// TIA Portal project "Custom_end_assignment" (V17)

(* hardware
DEVICE "S7-1200 station_1"  S7-1200 Station
   slot 0: "Rack_0"  S7-1200 Rack  Rack  V1.0
   slot 1: "PLC_1"  CPU 1215C AC/DC/Rly  6ES7 215-1BG40-0XB0  V4.5
DEVICE "HMI_1"  KTP700 Basic PN
   slot 0: "HMI_1"  KTP700 Basic PN  6AV2 123-2GB03-0AX0  17.0.0.0
   slot 1: "HMI_RT_1"  KTP700 Basic PN  6AV2 123-2GB03-0AX0  17.0.0.0
   slot 5: "HMI_1.IE_CP_1"  PROFINET Interface  17.0.0.0
      slot 1: "PROFINET Interface_1"  PROFINET Interface
         slot 1: "Port_1"  Port
*)

// ===== PLC "PLC_1"  CPU 1215C AC/DC/Rly =====

VAR_GLOBAL   // PLC tag table "Default tag table"
   "System_Byte" AT %MB1 : Byte;
   "FirstScan" AT %M1.0 : Bool;
   "DiagStatusUpdate" AT %M1.1 : Bool;
   "AlwaysTRUE" AT %M1.2 : Bool;
   "AlwaysFALSE" AT %M1.3 : Bool;
   "Clock_Byte" AT %MB0 : Byte;
   "Clock_10Hz" AT %M0.0 : Bool;
   "Clock_5Hz" AT %M0.1 : Bool;
   "Clock_2.5Hz" AT %M0.2 : Bool;
   "Clock_2Hz" AT %M0.3 : Bool;
   "Clock_1.25Hz" AT %M0.4 : Bool;
   "Clock_1Hz" AT %M0.5 : Bool;
   "Clock_0.625Hz" AT %M0.6 : Bool;
   "Clock_0.5Hz" AT %M0.7 : Bool;
END_VAR

VAR_GLOBAL   // PLC tag table "Hardware_I_O_Tags"
   "i_DR1_FlowSensorWaste" AT %I0.0 : Bool;
   "i_DR2_FlowSensorProduct" AT %I0.1 : Bool;
   "i_DR3_FlowSensorCocoa" AT %I0.2 : Bool;
   "i_DR4_FlowSensorSugar" AT %I0.3 : Bool;
   "i_RP_Start" AT %I0.4 : Bool;
   "i_RP_CocoaMinus" AT %I0.5 : Bool;
   "i_RP_CocoaPlus" AT %I0.6 : Bool;
   "i_RP_SugarMinus" AT %I0.7 : Bool;
   "i_RP_SugarPlus" AT %I1.0 : Bool;
   "i_RP_AllMilk" AT %I1.1 : Bool;
   "i_CP_CleanMinus" AT %I1.2 : Bool;
   "i_CP_BatchesMinus" AT %I1.3 : Bool;
   "i_CP_BatchesPlus" AT %I1.4 : Bool;
   "i_CP_1Batch" AT %I1.5 : Bool;
   "i_Tank_HeaterFeedback" AT %I8.0 : Bool;
   "i_Tank_LevelLow" AT %I8.1 : Bool;
   "i_Tank_LevelMiddle" AT %I8.2 : Bool;
   "i_Tank_LevelHigh" AT %I8.3 : Bool;
   "i_CP_Start" AT %I8.4 : Bool;
   "o_Tank_ValveWaste" AT %Q0.0 : Bool;
   "o_Tank_ValveProduct" AT %Q0.1 : Bool;
   "o_Tank_ValveCocoa" AT %Q0.2 : Bool;
   "o_Tank_ValveSugar" AT %Q0.3 : Bool;
   "o_Tank_ValveMilk" AT %Q0.4 : Bool;
   "o_Tank_ValveWater" AT %Q0.5 : Bool;
   "o_RP_Started_LED" AT %Q0.6 : Bool;
   "o_RP_Cocoa_LED" AT %Q0.7 : Bool;
   "o_RP_Sugar_LED" AT %Q1.0 : Bool;
   "o_RP_AllMilk_LED" AT %Q1.1 : Bool;
   "o_Tank_LevelEmpty_LED" AT %Q12.0 : Bool;
   "o_Tank_LevelLow_LED" AT %Q12.1 : Bool;
   "o_Tank_LevelMiddle_LED" AT %Q12.2 : Bool;
   "o_Tank_LevelHigh_LED" AT %Q12.3 : Bool;
   "o_Tank_Heater" AT %Q12.4 : Bool;
   "o_Tank_Mixer" AT %Q12.5 : Bool;
   "ai_Tank_Level" AT %IW64 : Int;
   "TankLevelScaledValue" AT %MD0 : Real;
   "ai_Tank_Temperature" AT %IW66 : Int;
   "TankTemperatureScaledValue" AT %MD4 : Real;
END_VAR

DATA_BLOCK "DB_MixerTank"   // DB2
{ S7_Optimized_Access := 'TRUE' }
VERSION : 0.1
   VAR
      i_FlowRate : Real := 1.0;
      ai_TankVolume : Real;
      ScaledTankVolume : Real;
      i_StartProcess : Bool;
      i_EmergencyStopOK : Bool;
      BoosterPumpMultiplier : Real := 5.0;
      MixerTankCapacity : Real := 500.0;
   END_VAR
BEGIN
END_DATA_BLOCK

// folder: 01_Communication/HumanMachineInterface

DATA_BLOCK "DB_MixerTankSystem"   // DB15
{ S7_Optimized_Access := 'TRUE' }
VERSION : 0.1
   VAR
      Valve1 : Bool;   // 0= closed, 1 = open
      Valve2 : Bool;   // 0= closed, 1 = open
      Valve3 : Bool;   // 0= closed, 1 = open
      FlowValve1 : Real;   // The amount of flow through valve 1 (input), Max 10 in normal mode
      FlowValve2 : Real;   // The amount of flow through valve 2 (input) Max 10 in normal mode
      FlowValve3 : Real;   // The amount of flow through valve 3 (output) Max 10 in normal mode
      MotorFlowValve1 : Bool;   // 0 = off / 1 = on
      MotorFlowValve2 : Bool;   // 0 = off / 1 = on
      MotorFlowValve3 : Bool;   // 0 = off / 1 = on
      MotorMixer : Bool;   // 0 = off / 1 = on
      TimerMotorMixer : Time;   // Timer Motor mixer is on (s)
      SystemStatusTank : Int;   // user defined type
      SensorTankVolumeHigh : Bool;   // sensor tank volume high
      SensorTankVolumeMiddle : Bool;   // sensor tank volume middle
      SensorTankVolumeLow : Bool;   // sensor tank volume low
      SensorBottleClamped : Bool;   // bottle is clamped by cilinder (1 = clamped / 0 = not clamped)
      Temperature : Real;
      ModeTemperature : Bool;   // 0= Celcius / 1= Fahrenheit
      Heating : Bool;   // 0 = off / 1 = on
      VolumeTank : Real;   // Total volume in the tank (MAX500L)
      NumberOfBottles : Int;   // Number of Bottles that are filled (each bottle 250 mL)
      "Status System" : String;   // defines message as 'fill bottle', valve1 open, valve 2 open
      Startbutton : Bool;
      StopButton : Bool;
   END_VAR
BEGIN
END_DATA_BLOCK

DATA_BLOCK "DB_BottleConveyer"   // DB16
{ S7_Optimized_Access := 'TRUE' }
VERSION : 0.1
   VAR
      A1 : Bool;   // Main switch bottle conveyor
      A2 : Bool;   // Automatic start bottle conveyor
      M1 : Bool;   // On/Off bottle conveyor
      B1 : Bool;   // Sensor infeed bottle conveyor
      B2 : Bool;   // Sensor bottle present filling nozzle
      B3 : Bool;   // Sensor bottle present bottlecheck
      B4 : Bool;   // Sensor bottle filled bottlecheck
      B5 : Bool;   // Sensor outfeed bottle conveyor
      P1 : Bool;   // Status servo bottle clamping
      P2 : Bool;   // Status servo cap positioning
   END_VAR
BEGIN
END_DATA_BLOCK

// folder: 01_Communication/System1

DATA_BLOCK "PC_Communication_Tags_Sys1"   // DB100
{ S7_Optimized_Access := 'TRUE' }
VERSION : 0.1
   VAR
      ServoPower : Bool;   // On/Off: On the HMI there is a button what switches on and off the power of the connected Servo
      RunState : Bool;   // This tag is True when the state of the whole system is 'Run'
      StopState : Bool;   // This tag is True when the state of the whole system is 'Stop'
      EnableReceiveCommands : Bool;   // On/Off: On the HMI there is a button what switches on and off the communication service
      MotorActiveFwd : Bool;   // This tag is True when the connected Servo is moving forward
      MotorActiveRev : Bool;   // This tag is True when the connected Servo is moving reverse
      SystemReadyServoActions : Bool;   // Only when all conditions are met (like described in the assessment document) this tag is True
      StartServoActions : Bool;   // When this tag is True, the Servo sequence may start "at the other side"
      ServoActionsFinished : Bool;   // When the actions to be executed for the connected Servo are finished, this tag is True
      BottlePresentRobot : Bool;   // This tag is True when a bottle is present at the robot
      BottleFilled : Bool;   // This tag is True when a bottle is filled
      BottleNotFilled : Bool;   // This tag is True when a bittle is not filled
      HeartBeat : Bool;   // This is a "heart beat" signal what is toggeling state in 0.5Hz frequency
   END_VAR
BEGIN
END_DATA_BLOCK

// folder: 01_Communication/System2

DATA_BLOCK "PC_Communication_Tags_Sys2"   // DB101
{ S7_Optimized_Access := 'TRUE' }
VERSION : 0.1
   VAR
      ServoPower : Bool;   // On/Off: On the HMI there is a button what switches on and off the power of the connected Servo
      RunState : Bool;   // This tag is True when the state of the whole system is 'Run'
      StopState : Bool;   // This tag is True when the state of the whole system is 'Stop'
      EnableReceiveCommands : Bool;   // On/Off: On the HMI there is a button what switches on and off the communication service
      MotorActiveFwd : Bool;   // This tag is True when the connected Servo is moving forward
      MotorActiveRev : Bool;   // This tag is True when the connected Servo is moving reverse
      SystemReadyServoActions : Bool;   // Only when all conditions are met (like described in the assessment document) this tag is True
      StartServoActions : Bool;   // When this tag is True, the Servo sequence may start "at the other side"
      ServoActionsFinished : Bool;   // When the actions to be executed for the connected Servo are finished, this tag is True
      BottlePresentRobot : Bool;   // This tag is True when a bottle is present at the robot
      BottleFilled : Bool;   // This tag is True when a bottle is filled
      BottleNotFilled : Bool;   // This tag is True when a bittle is not filled
      HeartBeat : Bool;   // This is a "heart beat" signal what is toggeling state in 0.5Hz frequency
   END_VAR
BEGIN
END_DATA_BLOCK

// folder: 02_Unit_MixerTank

DATA_BLOCK "UnitControl_MixerTank_DB"   // DB5
{ S7_Optimized_Access := 'TRUE' }
VERSION : 0.1
// stored: InstanceOfName UnitControl_MixerTank
"UnitControl_MixerTank"
BEGIN
END_DATA_BLOCK

// folder: 02_Unit_MixerTank/EquipmentModule_00_TankVolume

DATA_BLOCK "DB_TankVolume"   // DB8
{ S7_Optimized_Access := 'TRUE' }
VERSION : 0.1
   VAR
      EM_TankVolume : Real;
      EM_TankCapacity : Real := 500.0;
   END_VAR
BEGIN
END_DATA_BLOCK

// folder: 02_Unit_MixerTank/EquipmentModule_01_FlowInput

DATA_BLOCK "EM_FlowInput_DB"   // DB9
{ S7_Optimized_Access := 'TRUE' }
VERSION : 0.1
// stored: InstanceOfName EM_FlowInput
"EM_FlowInput"
BEGIN
END_DATA_BLOCK

// folder: 02_Unit_MixerTank/Simulated_Volume

DATA_BLOCK "Sim_Volume_DB"   // DB1
{ S7_Optimized_Access := 'TRUE' }
VERSION : 0.1
// stored: InstanceOfName Sim_Volume
"Sim_Volume"
BEGIN
END_DATA_BLOCK

// folder: 02_Unit_MixerTank/Z_iDBs

DATA_BLOCK "iDB_UnitControl_MixerTank"   // DB3
{ S7_Optimized_Access := 'TRUE' }
VERSION : 0.1
// stored: InstanceOfName UnitControl_MixerTank
"UnitControl_MixerTank"
BEGIN
END_DATA_BLOCK

// folder: 03_Unit_BottleConveyor/Z_iDBs

DATA_BLOCK "iDB_UnitControl_BottleConveyor"   // DB4
{ S7_Optimized_Access := 'TRUE' }
VERSION : 0.1
// stored: InstanceOfName UnitControl_BottleConveyor
"UnitControl_BottleConveyor"
BEGIN
END_DATA_BLOCK

// folder: (top level)

ORGANIZATION_BLOCK "PC_DrinksProduction"   // OB1, LAD, ProgramCycle
TITLE = "Main Program Sweep (Cycle)"
{ S7_Optimized_Access := 'TRUE' }
VERSION : 0.1
   VAR_INPUT
      Initial_Call : Bool;   // Initial call of this OB
      Remanence : Bool;   // =True, if remanent data are available
   END_VAR
BEGIN

REGION Network 2
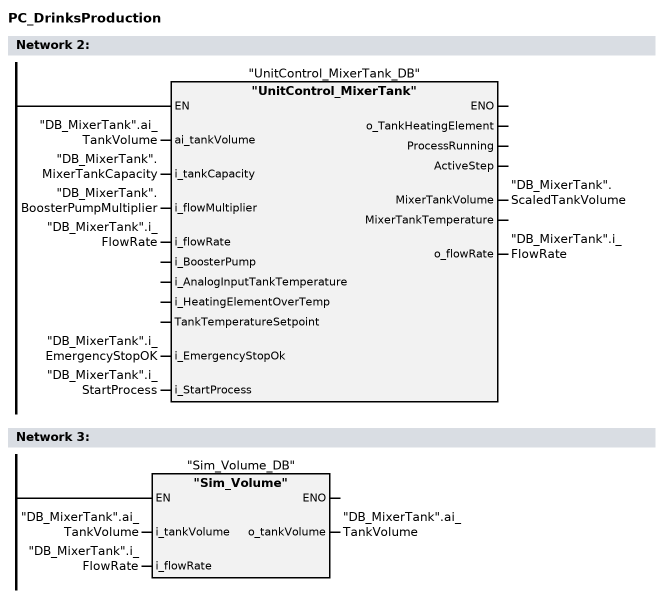
   RUNG wire#powerrail
      "UnitControl_MixerTank_DB"(ai_tankVolume := "DB_MixerTank".ai_TankVolume, i_tankCapacity := "DB_MixerTank".MixerTankCapacity, i_flowMultiplier := "DB_MixerTank".BoosterPumpMultiplier, i_flowRate := "DB_MixerTank".i_FlowRate, i_BoosterPump :=, i_AnalogInputTankTemperature :=, i_HeatingElementOverTemp :=, TankTemperatureSetpoint :=, i_EmergencyStopOk := "DB_MixerTank".i_EmergencyStopOK, i_StartProcess := "DB_MixerTank".i_StartProcess, o_TankHeatingElement =>, ProcessRunning =>, ActiveStep =>, MixerTankVolume => "DB_MixerTank".ScaledTankVolume, MixerTankTemperature =>, o_flowRate => "DB_MixerTank".i_FlowRate)
   END_RUNG
   // the same network as SCL:
   "UnitControl_MixerTank_DB"(ai_tankVolume := "DB_MixerTank".ai_TankVolume,   // "UnitControl_MixerTank"
                           i_tankCapacity := "DB_MixerTank".MixerTankCapacity,
                           i_flowMultiplier := "DB_MixerTank".BoosterPumpMultiplier,
                           i_flowRate := "DB_MixerTank".i_FlowRate,
                           i_EmergencyStopOk := "DB_MixerTank".i_EmergencyStopOK,
                           i_StartProcess := "DB_MixerTank".i_StartProcess,
                           MixerTankVolume => "DB_MixerTank".ScaledTankVolume,
                           o_flowRate => "DB_MixerTank".i_FlowRate);
END_REGION

REGION Network 3
   RUNG wire#powerrail
      "Sim_Volume_DB"(i_tankVolume := "DB_MixerTank".ai_TankVolume, i_flowRate := "DB_MixerTank".i_FlowRate, o_tankVolume => "DB_MixerTank".ai_TankVolume)
   END_RUNG
   // the same network as SCL:
   "Sim_Volume_DB"(i_tankVolume := "DB_MixerTank".ai_TankVolume,   // "Sim_Volume"
                   i_flowRate := "DB_MixerTank".i_FlowRate,
                   o_tankVolume => "DB_MixerTank".ai_TankVolume);
END_REGION
END_ORGANIZATION_BLOCK

// folder: 02_Unit_MixerTank

FUNCTION_BLOCK "UnitControl_MixerTank"   // FB2, LAD
TITLE = Unit mixer tank
{ S7_Optimized_Access := 'TRUE' }
VERSION : 0.1
   VAR_INPUT
      ai_tankVolume : Int;
      i_tankCapacity : Real;
      i_flowMultiplier : Real;
      i_flowRate : Real;
      i_BoosterPump : Bool;
      i_AnalogInputTankTemperature : Word;
      i_HeatingElementOverTemp : Bool;
      TankTemperatureSetpoint : Real;
      i_EmergencyStopOk : Bool;
      i_StartProcess : Bool;
   END_VAR
   VAR_OUTPUT
      o_TankHeatingElement : Bool;
      ProcessRunning : Bool;
      ActiveStep : Int;
      MixerTankVolume : Int;
      MixerTankTemperature : Real;
      o_flowRate : Real;
   END_VAR
   VAR
      iDB_EM_TankHeating : "EM_TankHeating";
      EnableHeating : Bool;
      msc_Heating : Bool;
      MixerTankSteps : Int;
      TankHeatingElementError : Bool;
      EM_TankVolume_Instance : "EM_TankVolume";
      TankVolume : Int;
   END_VAR
BEGIN

REGION Network 1 (SCL): Mixer tank stepper program
   // In this network the flowchart from your mixer tank process is translated to a so called " step program".
   CASE #MixerTankSteps OF
       0: // When PLC starts, Case is always 0
           #MixerTankSteps := 10;
       10:  // Initial step
           // used to reset / set to an initial state from your step program and all variables used in it.
           #ProcessRunning := FALSE;

           IF #i_EmergencyStopOk THEN 
               // Go to next step
               #MixerTankSteps := 20;
           END_IF;

       20: // Waiting for start process
           IF #i_StartProcess THEN
               #MixerTankSteps := 30;
           END_IF;

       30: // Fill tank with water
           // In teachers demo, the volume is read from the slider. 
           IF #TankVolume > 10.0 THEN
               #MixerTankSteps := 40;
           END_IF;

       40: // Start heating
           #EnableHeating := TRUE;
           IF NOT #TankHeatingElementError THEN
               #MixerTankSteps := 50;
           END_IF;

       50: // Waiting for level
           IF #TankVolume >= 100 THEN
               #MixerTankSteps := 60;
               ;
           END_IF;

       60:
           #EnableHeating := FALSE;
           IF #TankVolume <= 0.0 THEN
               // Statement section IF
               #MixerTankSteps := 10;
           END_IF;

       20..100:
           #ProcessRunning := TRUE;
           ;
       ELSE  // Statement section ELSE
           IF NOT #i_EmergencyStopOk THEN
               // Statement section IF
               #MixerTankSteps := 10;
               ;
           END_IF;
           ;
   END_CASE;
END_REGION

REGION Network 2: Minimum start conditions heater
   // To keep a structure in handling the minimum start conditions in a correct way all these conditions are commonly collected in one boolean, in this case called : msc_heating.
   // So: when this msc is false, under no condition the heater is enabled to start.
   // when this msc is true, the heater is allowed to start, when the stepper program gives it the command to do so.
   // 
   // In this case it is only the emergency stop circuit and the clixon " overheating check"  what can prevent the heater from starting
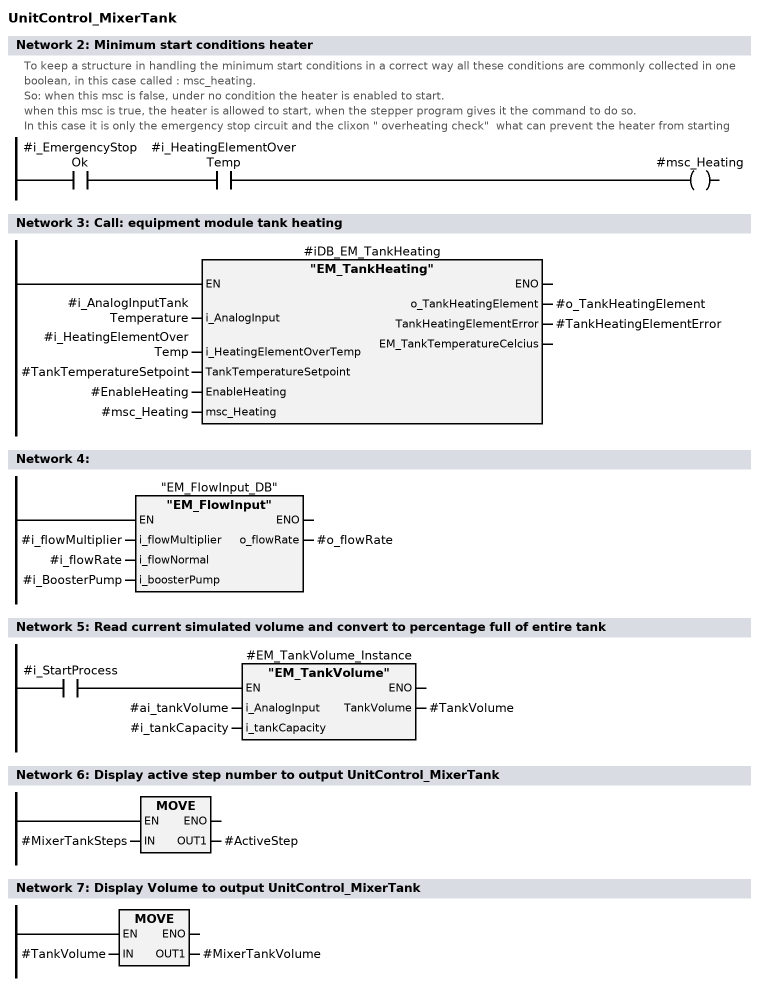
   RUNG wire#powerrail
      Contact( #i_EmergencyStopOk )
      Contact( #i_HeatingElementOverTemp )
      Coil( #msc_Heating )
   END_RUNG
   // the same network as SCL:
   #msc_Heating := #i_EmergencyStopOk AND #i_HeatingElementOverTemp;
END_REGION

REGION Network 3: Call: equipment module tank heating
   RUNG wire#powerrail
      #iDB_EM_TankHeating(i_AnalogInput := #i_AnalogInputTankTemperature, i_HeatingElementOverTemp := #i_HeatingElementOverTemp, TankTemperatureSetpoint := #TankTemperatureSetpoint, EnableHeating := #EnableHeating, msc_Heating := #msc_Heating, o_TankHeatingElement => #o_TankHeatingElement, TankHeatingElementError => #TankHeatingElementError, EM_TankTemperatureCelcius =>)
   END_RUNG
   // the same network as SCL:
   #iDB_EM_TankHeating(i_AnalogInput := #i_AnalogInputTankTemperature,   // "EM_TankHeating"
                       i_HeatingElementOverTemp := #i_HeatingElementOverTemp,
                       TankTemperatureSetpoint := #TankTemperatureSetpoint,
                       EnableHeating := #EnableHeating,
                       msc_Heating := #msc_Heating,
                       o_TankHeatingElement => #o_TankHeatingElement,
                       TankHeatingElementError => #TankHeatingElementError);
END_REGION

REGION Network 4
   RUNG wire#powerrail
      "EM_FlowInput_DB"(i_flowMultiplier := #i_flowMultiplier, i_flowNormal := #i_flowRate, i_boosterPump := #i_BoosterPump, o_flowRate => #o_flowRate)
   END_RUNG
   // the same network as SCL:
   "EM_FlowInput_DB"(i_flowMultiplier := #i_flowMultiplier,   // "EM_FlowInput"
                     i_flowNormal := #i_flowRate,
                     i_boosterPump := #i_BoosterPump,
                     o_flowRate => #o_flowRate);
END_REGION

REGION Network 5: Read current simulated volume and convert to percentage full of entire tank
   RUNG wire#powerrail
      Contact( #i_StartProcess )
      #EM_TankVolume_Instance(i_AnalogInput := #ai_tankVolume, i_tankCapacity := #i_tankCapacity, TankVolume => #TankVolume)
   END_RUNG
   // the same network as SCL:
   IF #i_StartProcess THEN
       #EM_TankVolume_Instance(i_AnalogInput := #ai_tankVolume,   // "EM_TankVolume"
                               i_tankCapacity := #i_tankCapacity,
                               TankVolume => #TankVolume);
   END_IF;
END_REGION

REGION Network 6: Display active step number to output UnitControl_MixerTank
   RUNG wire#powerrail
      Move(in := #MixerTankSteps, out1 => #ActiveStep)
   END_RUNG
   // the same network as SCL:
   #ActiveStep := #MixerTankSteps;
END_REGION

REGION Network 7: Display Volume to output UnitControl_MixerTank
   RUNG wire#powerrail
      Move(in := #TankVolume, out1 => #MixerTankVolume)
   END_RUNG
   // the same network as SCL:
   #MixerTankVolume := #TankVolume;
END_REGION

REGION Network 8: Dispaly Termperature to output UnitControl_MixerTank
END_REGION
END_FUNCTION_BLOCK

// folder: 02_Unit_MixerTank/EquipmentModule_00_TankVolume

FUNCTION_BLOCK "EM_TankVolume"   // FB4, FBD
TITLE = Equipment module tank volume
{ S7_Optimized_Access := 'TRUE' }
VERSION : 0.1
   VAR_INPUT
      i_AnalogInput : Real;
      i_tankCapacity : Real;
   END_VAR
   VAR_OUTPUT
      TankVolume : Real;
   END_VAR
BEGIN

REGION Network 1: Read Volume sensor from PLC hardware
   // WARNING: In this template, the analog sliders are used to determine the volume of the tank only for testing purposes! In the end assignment use case, the tank volume needs to be calculated!
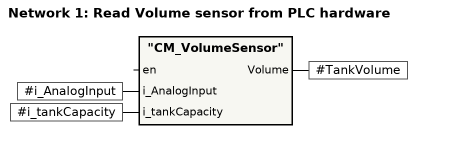
   "CM_VolumeSensor"(i_AnalogInput := #i_AnalogInput, i_tankCapacity := #i_tankCapacity, Volume => #TankVolume);
END_REGION
END_FUNCTION_BLOCK

// folder: 02_Unit_MixerTank/EquipmentModule_00_TankVolume/ControlModules

FUNCTION "CM_VolumeSensor" : Void   // FC3, LAD
TITLE = Read the volume sensor
{ S7_Optimized_Access := 'TRUE' }
VERSION : 0.1
// A fysical analog input is connected with a sensor what measures the height of the fluid level in the tank
   VAR_INPUT
      i_AnalogInput : Real;
      i_tankCapacity : Real;
   END_VAR
   VAR_OUTPUT
      Volume : Real;
   END_VAR
   VAR_TEMP
      NormValueVolumeInput : Real;
   END_VAR
BEGIN

REGION Network 1: Read analog input
   // Normalize analog input -> norm value (0.0 - 1.0)
   // Scale value to read the volume of a tank,
   // => scaling out a value for the tank is normalized from a volume of 0.0 (empty) to 100.0 procent (full).
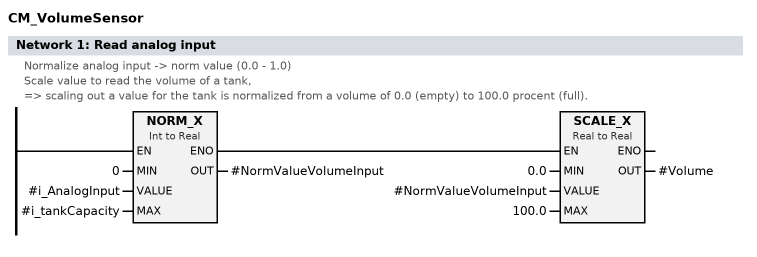
   RUNG wire#powerrail
      { S7_Templates := "[SrcType := Int, DestType := Real]" } Normalize(min := 0, value := #i_AnalogInput, max := #i_tankCapacity, out => #NormValueVolumeInput)
      { S7_Templates := "[SrcType := Real, DestType := Real]" } Scale(min := 0.0, value := #NormValueVolumeInput, max := 100.0, out => #Volume)
   END_RUNG
   // the same network as SCL:
   #NormValueVolumeInput := NORM_X(MIN := 0, VALUE := #i_AnalogInput, MAX := #i_tankCapacity);
   #Volume := SCALE_X(MIN := 0.0, VALUE := #NormValueVolumeInput, MAX := 100.0);
END_REGION
END_FUNCTION

// folder: 02_Unit_MixerTank/EquipmentModule_01_FlowInput

FUNCTION_BLOCK "EM_FlowInput"   // FB7, LAD
{ S7_Optimized_Access := 'TRUE' }
VERSION : 0.1
// determining the flow rate based on the booster pump status
   VAR_INPUT
      i_flowMultiplier : Real;
      i_flowNormal : Real;
      i_boosterPump : Bool;
   END_VAR
   VAR_OUTPUT
      o_flowRate : Real;
   END_VAR
BEGIN

REGION Network 1
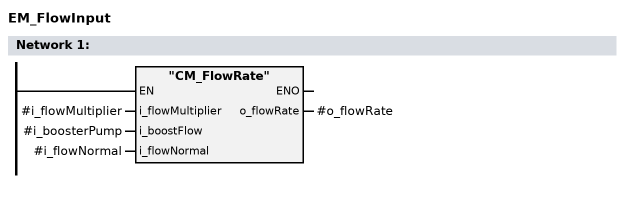
   RUNG wire#powerrail
      "CM_FlowRate"(i_flowMultiplier := #i_flowMultiplier, i_boostFlow := #i_boosterPump, i_flowNormal := #i_flowNormal, o_flowRate => #o_flowRate)
   END_RUNG
   // the same network as SCL:
   "CM_FlowRate"(i_flowMultiplier := #i_flowMultiplier,
                 i_boostFlow := #i_boosterPump,
                 i_flowNormal := #i_flowNormal,
                 o_flowRate => #o_flowRate);
END_REGION
END_FUNCTION_BLOCK

// folder: 02_Unit_MixerTank/EquipmentModule_01_FlowInput/ControlModules

FUNCTION "CM_FlowRate" : Void   // FC4, LAD
{ S7_Optimized_Access := 'TRUE' }
VERSION : 0.1
// Simulates the input flow of water into the tank, with the effects of the booster pump
   VAR_INPUT
      i_flowMultiplier : Real;
      i_boostFlow : Bool;
      i_flowNormal : Real;
   END_VAR
   VAR_OUTPUT
      o_flowRate : Real;
   END_VAR
   VAR_TEMP
      newFlow : Real;
   END_VAR
BEGIN

REGION Network 1
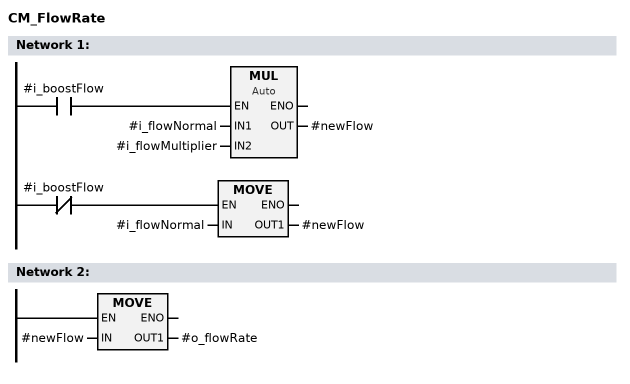
   RUNG wire#powerrail
      Contact( #i_boostFlow )
      Mul(in1 := #i_flowNormal, in2 := #i_flowMultiplier, out => #newFlow)
   END_RUNG
   RUNG wire#powerrail
      I_Contact( #i_boostFlow )
      Move(in := #i_flowNormal, out1 => #newFlow)
   END_RUNG
   // the same network as SCL:
   IF #i_boostFlow THEN #newFlow := #i_flowNormal * #i_flowMultiplier; END_IF;
   IF NOT #i_boostFlow THEN #newFlow := #i_flowNormal; END_IF;
END_REGION

REGION Network 2
   RUNG wire#powerrail
      Move(in := #newFlow, out1 => #o_flowRate)
   END_RUNG
   // the same network as SCL:
   #o_flowRate := #newFlow;
END_REGION
END_FUNCTION

// folder: 02_Unit_MixerTank/EquipmentModule_03_TankHeating

FUNCTION_BLOCK "EM_TankHeating"   // FB1, LAD
TITLE = Equipment module tank heating
{ S7_Optimized_Access := 'TRUE' }
VERSION : 0.1
// The equipment module tank heating takes control over the temperature from the tank by:
// - reading the actual temperature in the tank (slider on PLC-Sim)
// - reading the temperature setpoint from the HMI
// - Checking if the temperature from the heating element is not to high (checked by a clixon in the heating element).
// 
// The enabling of the heating element is done by the ...... Unit controlling the Equipment module heating.
   VAR_INPUT
      i_AnalogInput : Word;
      i_HeatingElementOverTemp : Bool;
      TankTemperatureSetpoint : Real;
      EnableHeating : Bool;
      msc_Heating : Bool;   // Minimum start conditions (like emergency stop)
   END_VAR
   VAR_OUTPUT
      o_TankHeatingElement : Bool;
      TankHeatingElementError : Bool;
      EM_TankTemperatureCelcius : Real;
   END_VAR
   VAR
      EnableHeatingElement : Bool;
      TankTemperatureCelcius : Real;
   END_VAR
BEGIN

REGION Network 1: Temperature control
   // Equipment module control tank heating
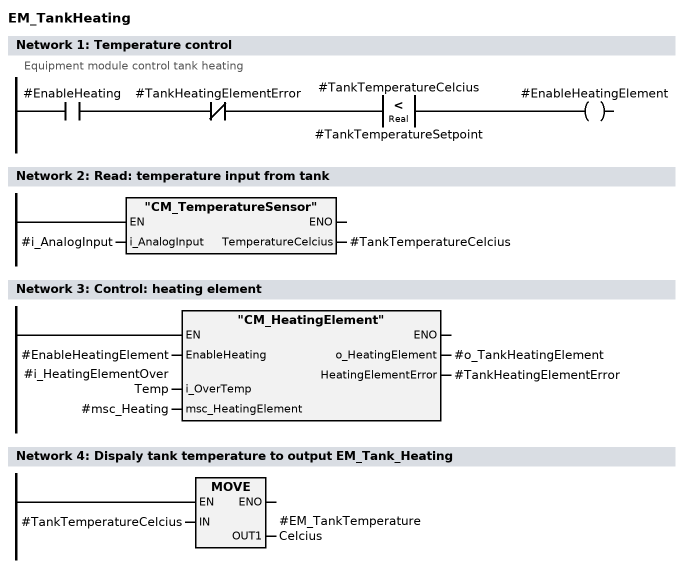
   RUNG wire#powerrail
      Contact( #EnableHeating )
      I_Contact( #TankHeatingElementError )
      { S7_Templates := "SrcType := Real" } LT_Contact(in1 := #TankTemperatureCelcius, in2 := #TankTemperatureSetpoint)
      Coil( #EnableHeatingElement )
   END_RUNG
   // the same network as SCL:
   #EnableHeatingElement := #EnableHeating AND NOT #TankHeatingElementError AND (#TankTemperatureCelcius < #TankTemperatureSetpoint);
END_REGION

REGION Network 2: Read: temperature input from tank
   RUNG wire#powerrail
      "CM_TemperatureSensor"(i_AnalogInput := #i_AnalogInput, TemperatureCelcius => #TankTemperatureCelcius)
   END_RUNG
   // the same network as SCL:
   "CM_TemperatureSensor"(i_AnalogInput := #i_AnalogInput, TemperatureCelcius => #TankTemperatureCelcius);
END_REGION

REGION Network 3: Control: heating element
   RUNG wire#powerrail
      "CM_HeatingElement"(EnableHeating := #EnableHeatingElement, i_OverTemp := #i_HeatingElementOverTemp, msc_HeatingElement := #msc_Heating, o_HeatingElement => #o_TankHeatingElement, HeatingElementError => #TankHeatingElementError)
   END_RUNG
   // the same network as SCL:
   "CM_HeatingElement"(EnableHeating := #EnableHeatingElement,
                       i_OverTemp := #i_HeatingElementOverTemp,
                       msc_HeatingElement := #msc_Heating,
                       o_HeatingElement => #o_TankHeatingElement,
                       HeatingElementError => #TankHeatingElementError);
END_REGION

REGION Network 4: Dispaly tank temperature to output EM_Tank_Heating
   RUNG wire#powerrail
      Move(in := #TankTemperatureCelcius, out1 => #EM_TankTemperatureCelcius)
   END_RUNG
   // the same network as SCL:
   #EM_TankTemperatureCelcius := #TankTemperatureCelcius;
END_REGION
END_FUNCTION_BLOCK

// folder: 02_Unit_MixerTank/EquipmentModule_03_TankHeating/ControlModules

FUNCTION "CM_TemperatureSensor" : Void   // FC1, LAD
TITLE = Tank temperature measurement
{ S7_Optimized_Access := 'TRUE' }
VERSION : 0.1
// A temperature sensor what is mounted in the bottom of the tank measures the temperature from the fluid in the tank.
   VAR_INPUT
      i_AnalogInput : Word;
   END_VAR
   VAR_OUTPUT
      TemperatureCelcius : Real;
   END_VAR
   VAR_TEMP
      NormValueTemperatureInput : Real;
   END_VAR
BEGIN

REGION Network 1: Read analog input
   // Normalize analog input -> norm value (0.0 - 1.0)
   // Scale value to readable temperature
   // => while we are measuring water containing fluid the temperature range can be between 0.0 degrees celcius and 100.0 degrees celcius
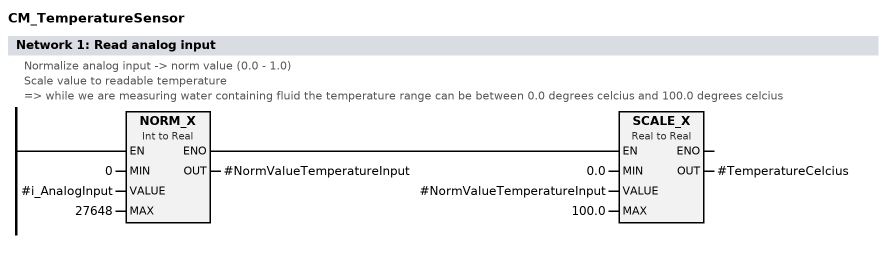
   RUNG wire#powerrail
      { S7_Templates := "[SrcType := Int, DestType := Real]" } Normalize(min := 0, value := #i_AnalogInput, max := 27648, out => #NormValueTemperatureInput)
      { S7_Templates := "[SrcType := Real, DestType := Real]" } Scale(min := 0.0, value := #NormValueTemperatureInput, max := 100.0, out => #TemperatureCelcius)
   END_RUNG
   // the same network as SCL:
   #NormValueTemperatureInput := NORM_X(MIN := 0, VALUE := #i_AnalogInput, MAX := 27648);
   #TemperatureCelcius := SCALE_X(MIN := 0.0, VALUE := #NormValueTemperatureInput, MAX := 100.0);
END_REGION
END_FUNCTION

FUNCTION "CM_HeatingElement" : Void   // FC2, FBD
{ S7_Optimized_Access := 'TRUE' }
VERSION : 0.1
   VAR_INPUT
      EnableHeating : Bool;
      i_OverTemp : Bool;   // 0= Heating element is overheated (detected by a "clixon"
      msc_HeatingElement : Bool;
   END_VAR
   VAR_OUTPUT
      o_HeatingElement : Bool;
      HeatingElementError : Bool;
   END_VAR
BEGIN

REGION Network 1: Control: heating element
   // When heating is enabled, heating element goes on
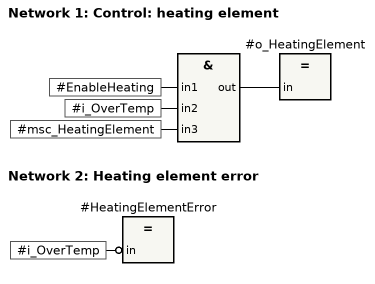
   #o_HeatingElement := #EnableHeating AND #i_OverTemp AND #msc_HeatingElement;
END_REGION

REGION Network 2: Heating element error
   // When the heating element is too hot, a clixon opens contact and generates error
   #HeatingElementError := NOT #i_OverTemp;
END_REGION
END_FUNCTION

// folder: 02_Unit_MixerTank/Simulated_Volume

FUNCTION_BLOCK "Sim_Volume"   // FB5, LAD
{ S7_Optimized_Access := 'TRUE' }
VERSION : 0.1
   VAR_INPUT
      i_tankVolume : Real;
      i_flowRate : Real;
   END_VAR
   VAR_OUTPUT
      o_tankVolume : Real;
   END_VAR
   VAR_TEMP
      pulseTrig : Bool;
   END_VAR
BEGIN

REGION Network 1
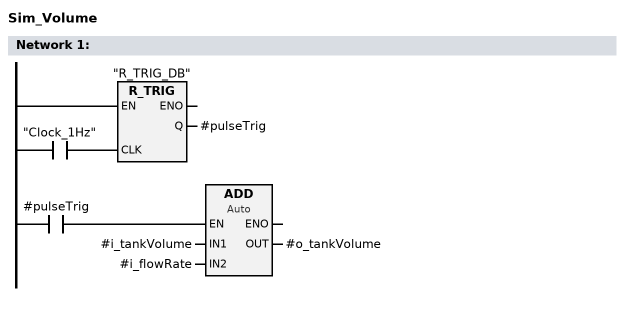
   "R_TRIG_DB"(CLK := "Clock_1Hz", Q => #pulseTrig);   // R_TRIG
   IF #pulseTrig THEN #o_tankVolume := #i_tankVolume + #i_flowRate; END_IF;
END_REGION
END_FUNCTION_BLOCK

// folder: 03_Unit_BottleConveyor

FUNCTION_BLOCK "UnitControl_BottleConveyor"   // FB3, FBD
{ S7_Optimized_Access := 'TRUE' }
VERSION : 0.1
BEGIN
END_FUNCTION_BLOCK

(* ===== HMI "HMI_RT_1" =====
system functions are stored by id; their names below are inferred from use
connection "HMI_Connection_1": ETHERNET, SMART_S7_1200_OMS

HMI tags "Default tag table"
   "Tag_ScreenNumber" : UInt, internal
   "DB_MixerTank_i_StartProcess" : Bool = PLC DB_MixerTank.i_StartProcess, 1 s
   "DB_MixerTank_i_EmergencyStopOK" : Bool = PLC DB_MixerTank.i_EmergencyStopOK, 1 s
   "DB_MixerTank_MixerTankCapacity" : Real = PLC DB_MixerTank.MixerTankCapacity, 1 s
   "DB_MixerTank_BoosterPumpMultiplier" : Real = PLC DB_MixerTank.BoosterPumpMultiplier, 1 s
   "DB_MixerTank_ScaledTankVolume" : Real = PLC DB_MixerTank.ScaledTankVolume, 1 s

Template "Template_1" 800x480
   Button "Exit" at 714,429 size 71x50; TextOff 'Exit'; PictureOff "ExitRuntime_KTP700_Basic_PN_TR"; PictureOn "ExitRuntime_KTP700_Basic_PN_TR"
      on Release: StopRuntime(0)
   Button "Template_Button" at 614,429 size 71x50; TextOff 'Text'
   Button "Template_Button_1" at 514,429 size 71x50; TextOff 'Text'
   Button "Template_Button_2" at 414,429 size 71x50; TextOff 'Text'
   Button "Template_Button_3" at 314,429 size 71x50; TextOff 'Text'
   Button "Template_Button_4" at 214,429 size 71x50; TextOff 'Text'
   Button "Alarms" at 114,429 size 71x50; TextOff 'Alarms'; PictureOff "AlarmDisplay_KTP700_Basic_PN_TR"; PictureOn "AlarmDisplay_KTP700_Basic_PN_TR"
      on Release: function_ef3f5d25("Alarm window_Unacknowledged", -1)
   Button "Start screen" at 14,429 size 71x50; TextOff 'Start screen'; PictureOff "NavigateHome_KTP700_Basic_PN_TR"; PictureOn "NavigateHome_KTP700_Basic_PN_TR"
   SymbolicIOField "Symbolic_IO_Field_Screen" at 93,9 size 600x33; TextOff '0'; TextOn '1'; TextList "TextList_ScreenNames"
      ProcessValue <- "Tag_ScreenNumber"
      on Change: ActivateScreenByNumber("Tag_ScreenNumber", 0)
   DateTimeField "HmiScreenItemData" at 695,25 size 105x25
   DateTimeField "HmiScreenItemData_1" at 695,0 size 105x25
   GraphicView "Logo" at 0,0 size 91x51; Picture "Logo of HMI_1"

screen "BottleConveyor Screen" 800x480
   on GenerateScreen: SetTag("Tag_ScreenNumber", 2)
   Button "HmiScreenItemData_1" at 269,26 size 211x47; TextOn 'Screen1'; TextOff 'BottleConveyor User Screen'; PictureOn "Navigates to Screen1 for KTP700 Basic+ PN 17.0.0.0"; PictureOff "Navigates to Screen0 for KTP700 Basic+ PN 17.0.0.0"
      on Release: ActivateScreen("BottleConveyor User Screen", 0)
   TextField "Text field_2" at 55,176 size 26x23; Text 'B1'
   TextField "Text field_4" at 378,204 size 26x23; Text 'B2'
   TextField "Text field_5" at 720,176 size 26x23; Text 'B5'
   TextField "Text field_8" at 593,225 size 26x23; Text 'B3'
   TextField "Text field_9" at 37,303 size 29x23; Text 'M1'
   TextField "Text field_10" at 78,359 size 144x23; Text 'Switches system'
   TextField "Text field_11" at 111,391 size 111x18; Text 'Main Switch (A1)'
   TextField "Text field_12" at 111,432 size 101x18; Text 'EmergencyStop'
   TextField "Text field_14" at 338,360 size 133x23; Text 'Automatic start'
   Switch "Switch_1" at 301,400 size 69x36; TextOn 'ON'; CaptionText 'Switch'; TextOff 'OFF'
   TextField "Text field_15" at 383,407 size 97x22; Text 'On/Off (A2)'
   TextField "Text field_27" at 593,200 size 26x23; Text 'B4'
   Switch "Switch_7" at 34,389 size 64x21; TextOn 'ON'; CaptionText 'Switch'; TextOff 'OFF'
   Switch "Switch_8" at 34,430 size 65x21; TextOn 'ON'; CaptionText 'Switch'; TextOff 'OFF'
   Group "Group" at 414,222 size 49x25
   Group "Group_1" at 316,222 size 49x25
   GraphicView "Graphic view_1" at 375,93 size 31x72; Picture "Graphic_13"
   TextField "Text field_6" at 274,108 size 96x23; Text 'Filling nozzle'
   Group "Group_2" at 254,175 size 57x51; Picture "Graphic_16"
   Group "Group_3" at 475,125 size 57x51; Picture "Graphic_16"
   TextField "Text field_13" at 546,395 size 159x22; Text 'Bottle clamping (P1)'
   TextField "Text field_16" at 546,430 size 158x22; Text 'Cap positioning (P2)'
   TextField "Text field_17" at 42,131 size 50x23; Text 'Infeed'
   TextField "Text field_18" at 707,131 size 61x23; Text 'Outfeed'
   TextField "Text field_19" at 625,360 size 57x23; Text 'Status'
   Group "Group_4" at 66,186 size 88x78; Picture "bottle_1"
   Button "HmiScreenItemData_2" at 32,26 size 157x47; TextOn 'Screen1'; TextOff 'MixerTank Screen'; PictureOn "Navigates to Screen1 for KTP700 Basic+ PN 17.0.0.0"; PictureOff "Navigates to Screen0 for KTP700 Basic+ PN 17.0.0.0"
      on Release: ActivateScreen("MixerTank Screen", 0)
   TextField "Text field_1" at 554,38 size 138x23; Text 'Conveyor Status'
   Group "Group_5" at 721,29 size 51x46; PictureOn "red_on"; PictureOff "red_off"
   GraphicView "Graphic view_3" at 254,197 size 57x29; Picture "Graphic_16"
   TextField "Text field_3" at 272,175 size 26x23; Text 'P1'
   GraphicView "Graphic view_4" at 475,147 size 57x29; Picture "Graphic_16"
   TextField "Text field_7" at 493,125 size 26x23; Text 'P2'
   Bar "Bar_1" at 96,205 size 28x56; MinimumValue 0; MaximumValue 100
   GraphicView "Graphic view_5" at 66,186 size 88x78; Picture "bottle_1"
   GraphicIOField "LED_STATUS_R" at 722,30 size 50x16; PictureOff "red_off"; PictureOn "red_on"
   GraphicIOField "LED_STATUS_Y" at 722,45 size 50x15; PictureOff "yellow_off"; PictureOn "yellow_on"
   GraphicIOField "LED_STATUS_G" at 722,60 size 50x15; PictureOff "green_off"; PictureOn "green_on"

screen "MixerTank Screen" 800x480
   on GenerateScreen: SetTag("Tag_ScreenNumber", 1)
   Button "HmiScreenItemData_2" at 24,28 size 186x47; TextOn 'Screen0'; TextOff 'MixerTank User Screen'; PictureOn "Navigates to Screen0 for KTP700 Basic+ PN 17.0.0.0"; PictureOff "Navigates to Screen0 for KTP700 Basic+ PN 17.0.0.0"
      on Release: ActivateScreen("MixerTank User Screen", 0)
   GraphicView "Graphic view_1" at 288,115 size 269x285; Picture "Graphic_18"
   GraphicView "Graphic view_8" at 431,182 size 52x41; Picture "Graphic_14"
   IOField "I/O field_1" at 325,182 size 96x32; FormatPattern s9999999999
   TextField "Text field_1" at 325,153 size 105x23; Text 'Timer mixer'
   TextField "Text field_5" at 582,167 size 98x23; Text 'Sensor Low'
   IOField "I/O field_4" at 389,348 size 75x32; FormatPattern s99999
   TextField "Text field_9" at 346,282 size 137x23; Text 'Heating ON/OFF'
   GraphicView "Graphic view_10" at 403,313 size 29x28; Picture "Graphic_22"
   IOField "I/O field_5" at 369,245 size 71x29; FormatPattern 999
   TextField "Text field_11" at 380,219 size 51x23; Text 'Temp'
   TextField "Text field_6" at 64,202 size 123x23; Text 'Controls Valve'
   IOField "I/O field_2" at 103,264 size 96x32; FormatPattern 999
   IOField "I/O field_7" at 103,310 size 96x32; FormatPattern 999
   IOField "I/O field_8" at 103,357 size 96x32; FormatPattern 999
   TextField "Text field_7" at 48,232 size 68x23; Text 'ON/OFF'
   TextField "Text field_12" at 33,264 size 15x23; Text '1'
   TextField "Text field_13" at 33,310 size 15x23; Text '2'
   TextField "Text field_14" at 33,357 size 15x23; Text '3'
   TextField "Text field_15" at 27,231 size 18x23; Text '#'
   TextField "Text field_16" at 660,168 size 102x23; Text 'Sensor High'
   TextField "Text field_17" at 660,201 size 119x23; Text 'Sensor Middle'
   TextField "Text field_18" at 660,233 size 98x23; Text 'Sensor Low'
   TextField "Text field_3" at 638,287 size 131x23; Text 'Bottle Clamped'
   TextField "Text field_4" at 48,144 size 149x23; Text 'MixerTank Status'
   TextField "Text field_10" at 593,134 size 160x23; Text 'Sensor information'
   IOField "I/O field_3" at 598,354 size 149x38; FormatPattern ??????????
   TextField "Text field_19" at 603,331 size 126x23; Text 'Status System'
   TextField "Text field_20" at 213,203 size 58x23; Text 'Motor'
   TextField "Text field_21" at 225,243 size 30x23; Text 'm1'
   TextField "Text field_22" at 225,291 size 30x23; Text 'm2'
   TextField "Text field_23" at 225,345 size 30x23; Text 'm3'
   TextField "Text field_8" at 332,390 size 153x23; Text 'Number of Bottles'
   TextField "Text field_24" at 325,219 size 34x23; Text 'C/F'
   TextField "Text field_25" at 439,153 size 51x23; Text 'Mixer'
   Bar "Bar_1" at 489,163 size 48x150; MinimumValue 0; MaximumValue 100
      ProcessValue <- "DB_MixerTank_ScaledTankVolume"
   TextField "Text field_2" at 505,140 size 16x23; Text 'V'
   Group "Group" at 208,126 size 61x54; PictureOn "red_on"; PictureOff "red_off"
   Button "HmiScreenItemData_1" at 593,28 size 186x47; TextOn 'Screen0'; TextOff 'BottleConveyer Screen'; PictureOn "Navigates to Screen0 for KTP700 Basic+ PN 17.0.0.0"; PictureOff "Navigates to Screen0 for KTP700 Basic+ PN 17.0.0.0"
      on Release: ActivateScreen("BottleConveyor Screen", 0)
   TextField "Text field_26" at 353,18 size 152x23; Text 'MixerTank Screen'
   GraphicIOField "LED_STATUS_R" at 209,127 size 60x19; PictureOn "red_on"; PictureOff "red_off"
   GraphicIOField "LED_STATUS_Y" at 209,145 size 60x18; PictureOn "yellow_on"; PictureOff "yellow_off"
   GraphicIOField "LED_STATUS_G" at 209,162 size 60x18; PictureOn "green_on"; PictureOff "green_off"

screen "ProcessCellDrinksProduction" 800x480, template "Template_1"
   on GenerateScreen: SetTag("Tag_ScreenNumber", 1)
   TextField "HmiScreenItemData_1" at 234,62 size 316x25; Text 'Process Cell Drinks production'
   Button "HmiScreenItemData" at 280,109 size 180x47; TextOn 'UnitServo'; TextOff 'BottleConveyor Screen'; PictureOn "Navigates to UnitServo for KTP700 Basic+ PN 17.0.0.0"; PictureOff "Navigates to UnitServo for KTP700 Basic+ PN 17.0.0.0"
      on Release: ActivateScreen("BottleConveyor Screen", 0)
   Button "HmiScreenItemData_3" at 94,109 size 180x47; TextOn 'Screen0'; TextOff 'MixerTank Screen'; PictureOn "Navigates to Screen0 for KTP700 Basic+ PN 17.0.0.0"; PictureOff "Navigates to Screen0 for KTP700 Basic+ PN 17.0.0.0"
      on Release: ActivateScreen("MixerTank Screen", 0)

screen "Project information" 800x480, template "Template_1"
   on GenerateScreen: SetTag("Tag_ScreenNumber", 5)
   TextField "HmiScreenItemData" at 107,102 size 171x28; Text 'Project name:'
   TextField "HmiScreenItemData_1" at 313,102 size 452x28; Text 'PC_LemonadeProcessing'
   TextField "HmiScreenItemData_2" at 107,132 size 171x28; Text 'Created on:'
   TextField "HmiScreenItemData_3" at 313,132 size 452x28; Text '12/22/2022 11:48:17 AM'
   TextField "HmiScreenItemData_4" at 107,162 size 171x28; Text 'Author:'
   TextField "HmiScreenItemData_5" at 313,162 size 452x28; Text '875361'
   TextField "HmiScreenItemData_6" at 107,192 size 171x28; Text 'Description:'
   TextField "HmiScreenItemData_7" at 313,192 size 452x28; Text 'Example project structure'
   Button "Back" at 73,52 size 159x47; TextOn 'Back'; TextOff 'Back'

screen "System information" 800x480, template "Template_1"
   on GenerateScreen: SetTag("Tag_ScreenNumber", 6)
   TextField "HmiScreenItemData" at 107,102 size 171x28; Text 'HMI device type:'
   TextField "HmiScreenItemData_1" at 313,102 size 452x28; Text 'KTP700 Basic+ PN 17.0.0.0'
   TextField "HmiScreenItemData_2" at 107,132 size 171x28; Text 'Connection:'
   TextField "HmiScreenItemData_3" at 313,132 size 452x28; Text '(not configured)'
   TextField "HmiScreenItemData_4" at 107,162 size 171x28; Text 'PLC:'
   TextField "HmiScreenItemData_5" at 313,162 size 452x28; Text '<PLC>'
   Button "Back" at 73,52 size 159x47; TextOn 'Back'; TextOff 'Back'

screen "MixerTank User Screen" 800x480
   Button "HmiScreenItemData_1" at 584,85 size 186x47; TextOn 'Screen0'; TextOff 'MixerTank Screen'; PictureOn "Navigates to Screen0 for KTP700 Basic+ PN 17.0.0.0"; PictureOff "Navigates to Screen0 for KTP700 Basic+ PN 17.0.0.0"
      on Release: ActivateScreen("MixerTank Screen", 0)
   Button "Button_1" at 583,177 size 156x66; TextOff 'Start Process'
      on Release: ActivateScreen("MixerTank Screen", 0); InvertBit("DB_MixerTank_i_StartProcess")
   Button "Button_2" at 584,289 size 200x175; TextOff 'Emergency Stop'
      on Release: InvertBit("DB_MixerTank_i_EmergencyStopOK")
   IOField "I/O field_1" at 334,324 size 54x34; FormatPattern s999999999.999
      ProcessValue <- "DB_MixerTank_MixerTankCapacity"
   TextField "Text field_1" at 85,335 size 167x23; Text 'MixerTank Capacity'
   TextField "Text field_2" at 85,394 size 202x23; Text 'Booster Pump Multiplier'
   IOField "I/O field_2" at 334,383 size 54x34; FormatPattern s999999999.999
      ProcessValue <- "DB_MixerTank_BoosterPumpMultiplier"
   TextField "Text field_3" at 166,264 size 114x23; Text 'User Settings'
   TextField "Text field_4" at 302,25 size 194x23; Text 'MixerTank User Screen'
   Button "HmiScreenItemData_2" at 31,85 size 186x47; TextOn 'Screen0'; TextOff 'System Overview'; PictureOn "Navigates to Screen0 for KTP700 Basic+ PN 17.0.0.0"; PictureOff "Navigates to Screen0 for KTP700 Basic+ PN 17.0.0.0"
      on Release: ActivateScreen("System Overview", 0)

screen "System Overview" 800x480
   Button "HmiScreenItemData_2" at 445,167 size 213x47; TextOn 'Screen0'; TextOff 'BottleConveyor User Screen'; PictureOn "Navigates to Screen0 for KTP700 Basic+ PN 17.0.0.0"; PictureOff "Navigates to Screen0 for KTP700 Basic+ PN 17.0.0.0"
      on Release: ActivateScreen("BottleConveyor User Screen", 0)
   Button "HmiScreenItemData_1" at 105,246 size 186x47; TextOn 'Screen0'; TextOff 'MixerTank Screen'; PictureOn "Navigates to Screen0 for KTP700 Basic+ PN 17.0.0.0"; PictureOff "Navigates to Screen0 for KTP700 Basic+ PN 17.0.0.0"
      on Release: ActivateScreen("MixerTank Screen", 0)
   Button "HmiScreenItemData_3" at 445,247 size 213x47; TextOn 'Screen0'; TextOff 'BottleConveyor Screen'; PictureOn "Navigates to Screen0 for KTP700 Basic+ PN 17.0.0.0"; PictureOff "Navigates to Screen0 for KTP700 Basic+ PN 17.0.0.0"
      on Release: ActivateScreen("BottleConveyor Screen", 0)
   Button "HmiScreenItemData_4" at 105,167 size 186x47; TextOn 'Screen0'; TextOff 'MixerTank User Screen'; PictureOn "Navigates to Screen0 for KTP700 Basic+ PN 17.0.0.0"; PictureOff "Navigates to Screen0 for KTP700 Basic+ PN 17.0.0.0"
      on Release: ActivateScreen("MixerTank User Screen", 0)
   TextField "Text field_1" at 153,87 size 86x23; Text 'SYSTEM 1'
   TextField "Text field_2" at 494,87 size 86x23; Text 'SYSTEM 2'

screen "BottleConveyor User Screen" 800x480
   Button "HmiScreenItemData_1" at 583,102 size 186x47; TextOn 'Screen0'; TextOff 'BottleConveyor Screen'; PictureOn "Navigates to Screen0 for KTP700 Basic+ PN 17.0.0.0"; PictureOff "Navigates to Screen0 for KTP700 Basic+ PN 17.0.0.0"
      on Release: ActivateScreen("BottleConveyor Screen", 0)
   Button "Button_3" at 584,184 size 156x66; TextOff 'Start Process'
   Button "Button_4" at 584,289 size 200x175; TextOff 'Emergency Stop'
   TextField "Text field_4" at 281,25 size 233x23; Text 'BottleConveyor User Screen'
   Button "HmiScreenItemData_2" at 26,102 size 186x47; TextOn 'Screen0'; TextOff 'System Overview'; PictureOn "Navigates to Screen0 for KTP700 Basic+ PN 17.0.0.0"; PictureOff "Navigates to Screen0 for KTP700 Basic+ PN 17.0.0.0"
      on Release: ActivateScreen("System Overview", 0)
*)